// ---- POUs/XTS/Movers/VI_MoverVisu.TcVIS
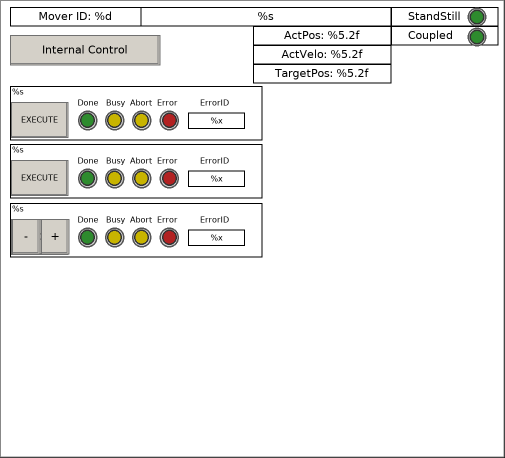
VISUALIZATION VI_MoverVisu  // 505x458
VAR_IN_OUT
	fbMover : FB_Mover;
END_VAR
    Rectangle (0,0 505x458)
    Rectangle (140,7 251x19), "%s", text variable: fbMover.ax.Status.MotionState, text list: 'AxisState_txt'
    Frame (10,86 252x54)
        shows VI_PLCOpenState(bExecute := fbMover.fbPower.Enable, sName := 'Power', bBusy := fbMover.fbPower.Busy, bDone := fbMover.fbPower.Status, bError := fbMover.fbPower.Error, bCommandAborted := fbMover.bTmp, ErrorID := fbMover.fbPower.ErrorID)
    Frame (10,144 252x54)
        shows VI_PLCOpenState(bExecute := fbMover.fbReset.Execute, sName := 'Reset', bBusy := fbMover.fbReset.Busy, bDone := fbMover.fbReset.Done, bError := fbMover.fbReset.Error, bCommandAborted := fbMover.bTmp, ErrorID := fbMover.fbReset.ErrorId)
    Button (10,35 150x30), "Internal Control", tooltip "Enable Visu Control, all methods will be locked"
        toggle fbMover.bInternalControl
    Rectangle (391,7 107x19), "StandStill"
    Lamp1 (466,6 22x22), variable: fbMover.ax.Status.StandStill, style: Lamp-Lamp1-Green
    Rectangle (10,7 131x19), "Mover ID: %d", text variable: fbMover.udiID
    Rectangle (253,26 138x19), "ActPos: %5.2f", text variable: fbMover.ax.NcToPlc.ModuloActPos, text list: 'AxisState_txt'
    Rectangle (253,45 138x19), "ActVelo: %5.2f", text variable: fbMover.ax.NcToPlc.ActVelo, text list: 'AxisState_txt'
    Rectangle (391,26 107x19), "Coupled"
    Lamp1 (466,26 22x22), variable: fbMover.ax.Status.Coupled, style: Lamp-Lamp1-Green
    Frame (10,203 252x54)
        shows VI_PLCOpenState(bExecute := fbMover.bTmp, sName := 'JogCA', bBusy := fbMover.fbJogCA.Busy, bDone := fbMover.fbJogCA.Done, bError := fbMover.fbJogCA.Error, bCommandAborted := fbMover.fbJogCA.CommandAborted, ErrorID := fbMover.fbJogCA.ErrorID)
    Button (12,219 28x35), "-"
        toggle fbMover.fbJogCA.JogBackwards
    Button (41,219 28x35), "+"
        toggle fbMover.fbJogCA.JogForward
    Rectangle (253,64 138x19), "TargetPos: %5.2f", text variable: fbMover.lrTargetPos, text list: 'AxisState_txt'
END_VISUALIZATION

// ---- POUs/XTS/Movers/VI_MoversVisu.TcVIS
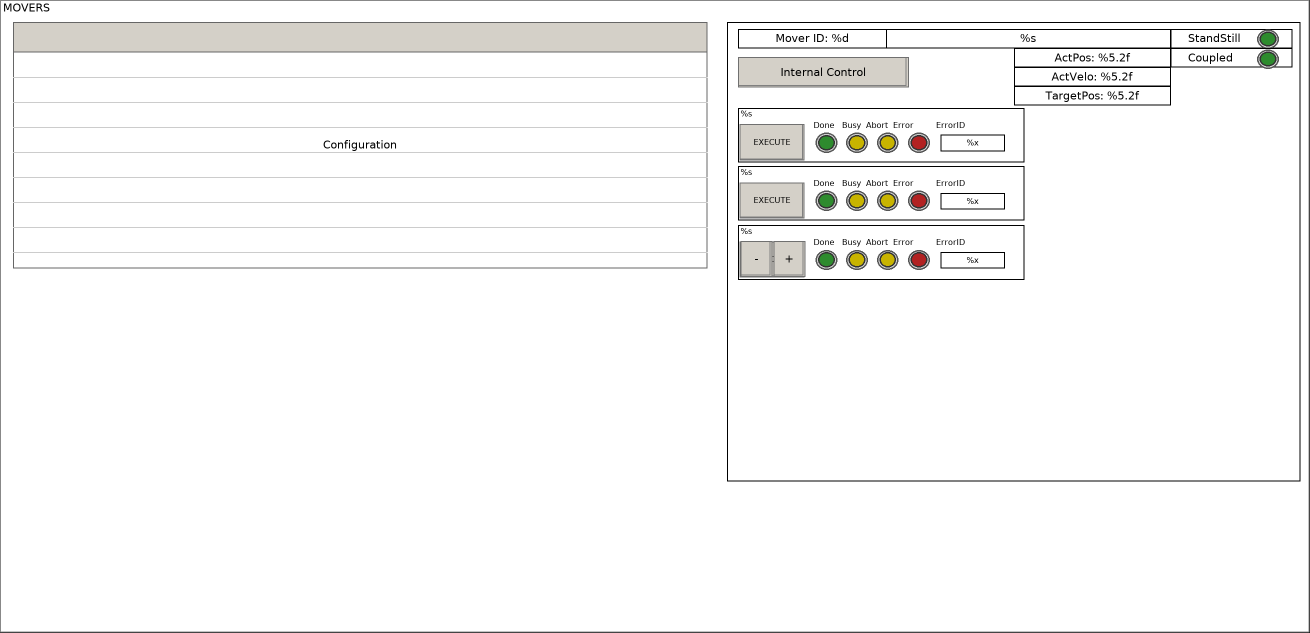
VISUALIZATION VI_MoversVisu  // 1310x633
VAR_IN_OUT
	ax		: ARRAY [1..Tc3_XTS_Utility.TcIoXtsEnvironmentParameterList.MaxXtsMoversPerXpu] OF FB_Mover;
END_VAR
VAR
	stTableStruct : ARRAY [1..25] OF stTableStructx10;
	iSelectedMover : INT;
END_VAR
    Rectangle (0,0 1310x633), "MOVERS"
    Frame (727,22 573x459), frame switch variable: iSelectedMover-1
        shows VI_MoverVisu(fbMover := ax[1])
        shows VI_MoverVisu(fbMover := ax[2])
        shows VI_MoverVisu(fbMover := ax[3])
        shows VI_MoverVisu(fbMover := ax[4])
        shows VI_MoverVisu(fbMover := ax[5])
        shows VI_MoverVisu(fbMover := ax[6])
        shows VI_MoverVisu(fbMover := ax[7])
        shows VI_MoverVisu(fbMover := ax[8])
        shows VI_MoverVisu(fbMover := ax[9])
        shows VI_MoverVisu(fbMover := ax[10])
        shows VI_MoverVisu(fbMover := ax[11])
        shows VI_MoverVisu(fbMover := ax[12])
        shows VI_MoverVisu(fbMover := ax[13])
        shows VI_MoverVisu(fbMover := ax[14])
        shows VI_MoverVisu(fbMover := ax[15])
        shows VI_MoverVisu(fbMover := ax[16])
        shows VI_MoverVisu(fbMover := ax[17])
        shows VI_MoverVisu(fbMover := ax[18])
        shows VI_MoverVisu(fbMover := ax[19])
        shows VI_MoverVisu(fbMover := ax[20])
        shows VI_MoverVisu(fbMover := ax[21])
        shows VI_MoverVisu(fbMover := ax[22])
        shows VI_MoverVisu(fbMover := ax[23])
        shows VI_MoverVisu(fbMover := ax[24])
        shows VI_MoverVisu(fbMover := ax[25])
    Table (13,22 694x246), "Configuration", data array: stTableStruct
        p1137915858: iSelectedMover
        p3854506369: ax[INDEX].ax.NcToPlc.AxisId
        p1892666644: ax[INDEX].ax.NcToPlc.ModuloSetPos
        p338671338: ax[INDEX].ax.NcToPlc.SetVelo
        p2170511999: ax[INDEX].ax.Status.MotionState
        p3723444502: ax[INDEX].ax.NcToPlc.ErrorCode
        p511219082: Position
        p1755163831: Velocity
        p2237128397: Error ID
        p505689113: Process Time
        p1757482276: Stop Positions
        p4088588272: Ack Mode
        p2243050616: Disable
        p516019884: Travel Time
        p2685023577: stTableStruct.b1
        p3312258591: stTableStruct.b2
        p1791247317: stTableStruct.b3
        p262371475: stTableStruct.b4
        p4008173056: stTableStruct.b5
        p2340480326: stTableStruct.b6
        p606709900: stTableStruct.b7
        p1095668682: stTableStruct.b8
        p1037165547: stTableStruct.b9
        p1488378029: stTableStruct.b10
        Columns.Column.[8].Template: xts.aStations[INDEX].stCfg.bDisable=true; toggle xts.aStations[INDEX].stCfg.bDisable
        Columns.Column.[6].Template: OnMouseClick: write the text variable via Default, min 1, max 3
        Columns.Column.[4].Template: OnMouseClick: write the text variable via Default
        Columns.Column.[5].Template: OnMouseClick: write the text variable via Default
        Columns.Column.[7].Template: OnMouseClick: write the text variable via Default
        Columns.Column.[9].Template: OnMouseClick: write the text variable via Default
END_VISUALIZATION

// ---- POUs/XTS/Stations/VI_StationVISU.TcVIS
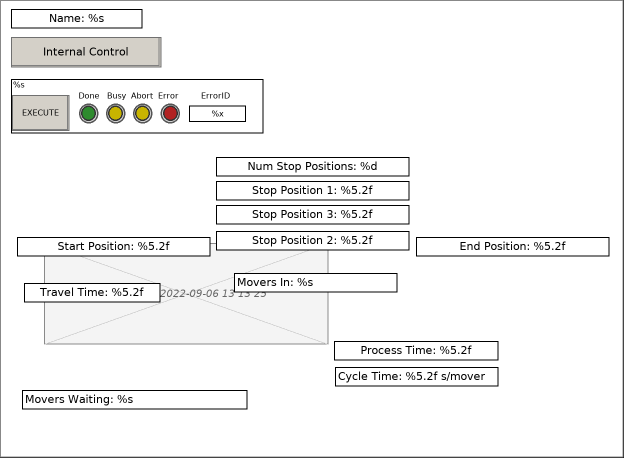
VISUALIZATION VI_StationVISU  // 624x458
VAR_IN_OUT
	fbStation : FB_Station;
END_VAR
    Rectangle (0,0 624x458)
    Frame (11,79 252x54)
        shows VI_PLCOpenState(bExecute := fbStation.bStart, sName := 'Secuence', bBusy := fbStation.stSecuenceStatus.bBusy, bDone := fbStation.stSecuenceStatus.bDone, bError := fbStation.stSecuenceStatus.bError, ErrorID := fbStation.stSecuenceStatus.udiErrorID)
    Button (11,37 150x30), "Internal Control", tooltip "Enable Visu Control, all methods will be locked"
        toggle fbStation.bInternalControl
    Rectangle (11,9 131x19), "Name: %s", text variable: fbStation.stCfg.sName
        OnMouseClick: write the text variable via Default
    Image (44,243 284x101), image: ImagePool.2022-09-06 13 13 25
    Rectangle (17,237 193x19), "Start Position: %5.2f", text variable: fbStation.stCfg.lrStartPosition
        OnMouseClick: write the text variable via Default
    Rectangle (416,237 193x19), "End Position: %5.2f", text variable: fbStation.stCfg.lrEndPosition
        OnMouseClick: write the text variable via Default
    Rectangle (234,273 163x19), "Movers In: %s", text variable: fbStation.sMoversIn
        OnMouseClick: write the text variable via Default
    Rectangle (22,390 225x19), "Movers Waiting: %s", text variable: fbStation.sMoversWaiting
        OnMouseClick: write the text variable via Default
    Rectangle (216,157 193x19), "Num Stop Positions: %d", text variable: fbStation.stCfg.uiNumStopPositions
        OnMouseClick: write the text variable via Default
    Rectangle (216,181 193x19), "Stop Position 1: %5.2f", text variable: fbStation.stCfg.lrStopPosition[1]
        OnMouseClick: write the text variable via Default
    Rectangle (216,231 193x19), "Stop Position 2: %5.2f", text variable: fbStation.stCfg.lrStopPosition[2], invisible if: fbStation.stCfg.uiNumStopPositions < 2
        OnMouseClick: write the text variable via Default
    Rectangle (216,205 193x19), "Stop Position 3: %5.2f", text variable: fbStation.stCfg.lrStopPosition[3], invisible if: fbStation.stCfg.uiNumStopPositions < 3
        OnMouseClick: write the text variable via Default
    Rectangle (335,367 163x19), "Cycle Time: %5.2f s/mover", text variable: (fbStation.lrActualProcessTime+fbStation.lrActualWaitingTime)/udint_to_lreal(fbStation.stCfg.uiNumStopPositions)
    Rectangle (24,283 136x19), "Travel Time: %5.2f", text variable: fbStation.stCfg.lrTravelTime
        OnMouseClick: write the text variable via Default
    Rectangle (334,341 164x19), "Process Time: %5.2f", text variable: fbStation.stCfg.lrProcessingTime
        OnMouseClick: write the text variable via Default
END_VISUALIZATION

// ---- POUs/XTS/Stations/VI_StationsVISU.TcVIS
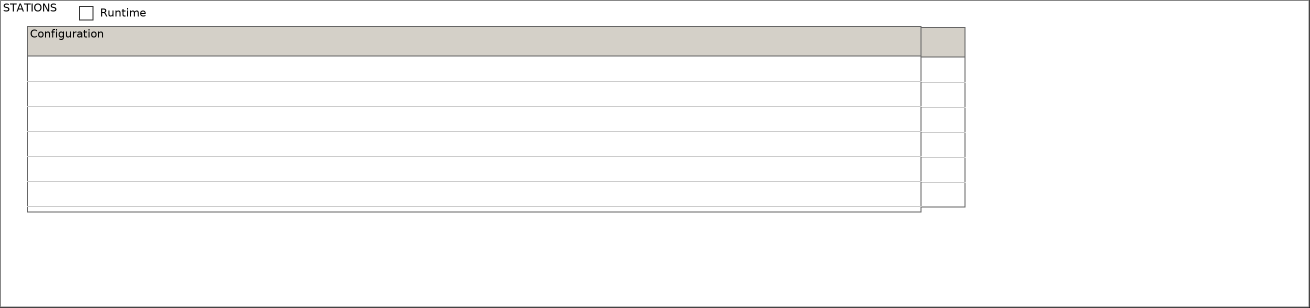
VISUALIZATION VI_StationsVISU  // 1310x308
VAR_IN_OUT
	aStations		: ARRAY [1..Tc3_XTS_Utility.TcIoXtsEnvironmentParameterList.MaxXtsInfoStation] OF FB_Station; //Stations
END_VAR
VAR
	stTableStruct : ARRAY [1..25] OF stTableStructx10;
	iSelectedStation : INT;
	bRunTime		: BOOL;
END_VAR
    Rectangle (0,0 1310x308), "STATIONS"
    Table (27,27 938x180), "Configuration", invisible if: bRunTime=true, data array: stTableStruct
        p1137915858: iSelectedStation
        p3854506369: aStations[INDEX].stCfg.sName
        p1892666644: aStations[INDEX].stCfg.lrStartPosition
        p338671338: aStations[INDEX].stCfg.lrStopPosition[1]
        p2170511999: aStations[INDEX].stCfg.lrStopPosition[2]
        p3723444502: aStations[INDEX].stCfg.lrStopPosition[3]
        p1218418051: aStations[INDEX].stCfg.lrProcessingTime
        p746581629: aStations[INDEX].stCfg.uiNumStopPositions
        p3104783080: aStations[INDEX].stCfg.lrTravelTime
        p7306298: aStations[INDEX].stCfg.lrEndPosition
        p511219082: Start Position
        p1755163831: Stop Position 1
        p4092479075: Stop Position 2
        p2237128397: Stop Position 3
        p505689113: Process Time
        p1757482276: Stop Positions
        p4088588272: Travel Time
        p2243050616: Extra Cfg.
        p516019884: End Position
        p2685023577: stTableStruct.b1
        p3312258591: stTableStruct.b2
        p1791247317: stTableStruct.b3
        p262371475: stTableStruct.b4
        p4008173056: stTableStruct.b5
        p2340480326: stTableStruct.b6
        p606709900: stTableStruct.b7
        p1095668682: stTableStruct.b8
        p1037165547: stTableStruct.b9
        p1488378029: stTableStruct.b10
        Columns.Column.[3].Template: OnMouseClick: write the text variable via Default
        Columns.Column.[6].Template: OnMouseClick: write the text variable via Default, min 1, max 3
        Columns.Column.[4].Template: OnMouseClick: write the text variable via Default
        Columns.Column.[5].Template: OnMouseClick: write the text variable via Default
        Columns.Column.[2].Template: OnMouseClick: write the text variable via Default
        Columns.Column.[7].Template: OnMouseClick: write the text variable via Default
        Columns.Column.[9].Template: OnMouseClick: write the text variable via Default
        Columns.Column.[1].Template: OnMouseClick: write the text variable via Default
    Checkbox (77,2 150x22), "Runtime", variable: bRunTime
    Table (27,26 894x186), "Configuration", invisible if: bRunTime=false, data array: stTableStruct
        p225073791: %5.2f s/m
        p3854506369: aStations[INDEX].stCfg.sName
        p1892666644: aStations[INDEX].stCfg.bEnableManualAck
        p338671338: aStations[INDEX].stCfg.bManualAck
        p2170511999: aStations[INDEX].fbMoversFIFO.nMovers
        p3723444502: aStations[INDEX].stCfg.udiSequenceState
        p1218418051: aStations[INDEX].udiErrorID
        p746581629: aStations[INDEX].sMoversWaiting
        p3104783080: aStations[INDEX].sMoversIn
        p2501879983: (aStations[INDEX].lrActualProcessTime+aStations[INDEX].lrActualWaitingTime)/udint_to_lreal(aStations[INDEX].stCfg.uiNumStopPositions)
        p7306298: xts.aStations[INDEX].lrActualWaitingTime
        p511219082: M. Ack
        p4092479075: Movers Waiting
        p505689113: Error ID
        p4088588272: Movers In
        p2243050616: Cycle Time
        p516019884: Waiting Time
        p2685023577: stTableStruct.b1
        p3312258591: stTableStruct.b2
        p1791247317: stTableStruct.b3
        p262371475: stTableStruct.b4
        p4008173056: stTableStruct.b5
        p2340480326: stTableStruct.b6
        p606709900: stTableStruct.b7
        p1095668682: stTableStruct.b8
        p1037165547: stTableStruct.b9
        p1488378029: stTableStruct.b10
        Columns.Column.[6].Template: OnMouseClick: write the text variable via Default, min 1, max 3
        Columns.Column.[4].Template: OnMouseClick: write the text variable via Default
        Columns.Column.[5].Template: OnMouseClick: write the text variable via Default
        Columns.Column.[2].Template: tap aStations[INDEX].stCfg.bManualAck
        Columns.Column.[0].Template: OnMouseClick: write the text variable via Default
        Columns.Column.[7].Template: OnMouseClick: write the text variable via Default
        Columns.Column.[9].Template: OnMouseClick: write the text variable via Default
        Columns.Column.[1].Template: toggle aStations[INDEX].stCfg.bEnableManualAck
END_VISUALIZATION

// ---- POUs/XTS/VISUs/TextList/AxisState_txt.TcTLO
TEXTLIST AxisState_txt
  0 = 'INVALID'
  1 = 'DISABLED'
  2 = 'STANDSTILL'
  3 = 'ERROR STOP'
  4 = 'STOPPING'
  5 = 'HOMING'
  6 = 'DISCRETE MOTION'
  7 = 'CONTINIOUS MOTION'
  8 = 'SYNCHRONIZED MOTION'
   = ''
END_TEXTLIST

// ---- POUs/XTS/VISUs/TextList/GroupState_txt.TcTLO
TEXTLIST GroupState_txt
  0 = 'INVALID'
  1 = 'DISABLED'
  2 = 'STANDBY'
  3 = 'MOVING'
  4 = 'STOPPING'
  5 = 'ERROR STOP'
  6 = 'HOMING'
  7 = 'NOT READY'
  8 = 'SUSPENDED'
   = ''
END_TEXTLIST

// ---- POUs/XTS/VISUs/TextList/MoversMode_txt.TcTLO
TEXTLIST MoversMode_txt
  1 = 'Single'
  2 = 'Double'
  3 = 'Triple'
   = ''
END_TEXTLIST

// ---- POUs/XTS/VISUs/TextList/PML_Modes_txt.TcTLO
TEXTLIST PML_Modes_txt
  0 = 'Undefined'
  1 = 'Production'
  2 = 'Manual'
   = ''
END_TEXTLIST

// ---- POUs/XTS/VISUs/VI_PLCOpenState.TcVIS
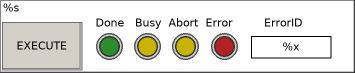
VISUALIZATION VI_PLCOpenState  // 355x73
VAR_IN_OUT
	bExecute : BOOL;	
END_VAR
VAR_INPUT
	sName	: STRING;
	bBusy : BOOL;
	bDone : BOOL;
	bError: BOOL;
	bCommandAborted : BOOL;
	ErrorID:UDINT;
END_VAR
    Rectangle (0,0 355x73), "%s", text variable: sName
    Lamp1 (94,31 31x31), variable: bDone, style: Lamp-Lamp1-Green
    Lamp1 (132,31 31x31), variable: bBusy, style: Lamp-Lamp1-Yellow
    Lamp1 (170,31 31x31), variable: bCommandAborted, style: Lamp-Lamp1-Yellow
    Lamp1 (209,31 31x31), variable: bError, style: Lamp-Lamp1-Red
    Rectangle (251,36 80x22), "%x", text variable: ErrorID
    Label (75,8 271x30), "Done Busy Abort Error ErrorID"
    Button (2,22 80x48), "EXECUTE"
        toggle bExecute
END_VISUALIZATION

// ---- POUs/XTS/VISUs/VI_XTSManualVisu.TcVIS
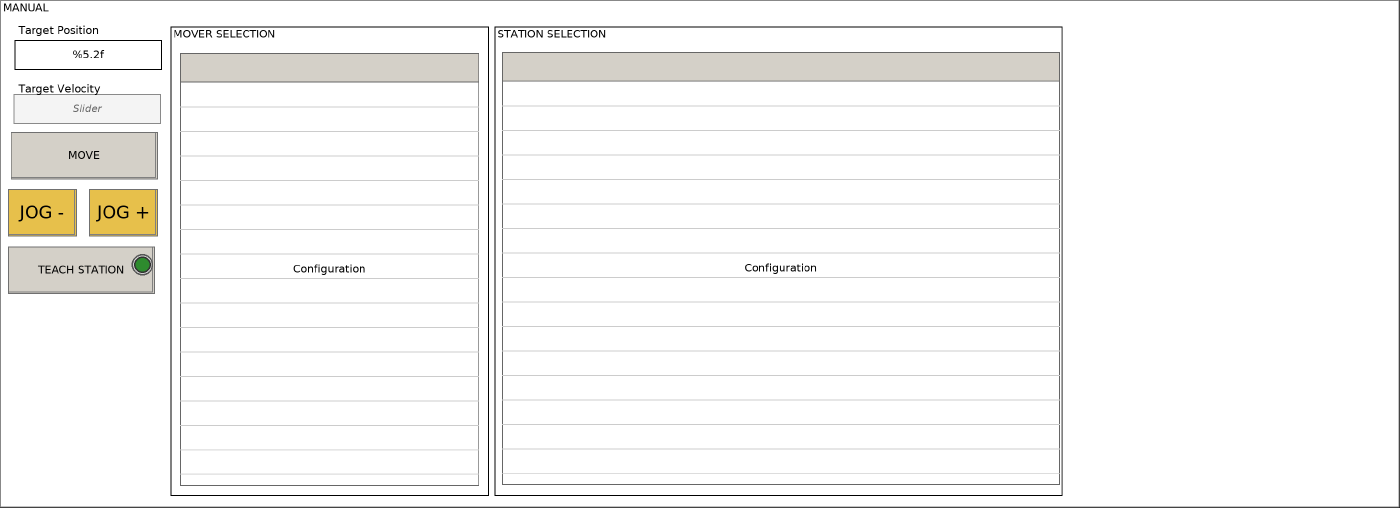
VISUALIZATION VI_XTSManualVisu  // 1430x519
VAR_IN_OUT
	xts : XTS_System;
END_VAR
VAR
	stTableStruct : ARRAY [1..20] OF stTableStructx10;
END_VAR
    Rectangle (0,0 1430x519), "MANUAL"
    Button (11,135 150x48), "MOVE"
        tap xts.bManualMove
    Slider (14,96 150x30), variable: xts.lrTargetVelocity, scale 1..4000
    Label (16,76 150x30), "Target Velocity"
    Rectangle (15,41 150x30), "%5.2f", text variable: xts.lrTargetPosition, input disabled if: xts.udiStationSelection<>0
        OnMouseClick: write the text variable via Default
    Label (16,16 150x30), "Target Position"
    Button (8,252 150x48), "TEACH STATION", input disabled if: xts.iVisuMoverSelection<1
        tap xts.bTeachStation
    Lamp1 (133,256 25x29), variable: xts.bTeachDone, style: Lamp-Lamp1-Green
    Rectangle (174,27 325x479), "MOVER SELECTION"
    Table (184,54 305x442), "Configuration", data array: stTableStruct
        p1137915858: xts.iVisuMoverSelection
        p3854506369: xts.ax[INDEX].ax.NcToPlc.AxisId
        p1892666644: xts.ax[INDEX].ax.NcToPlc.ModuloSetPos
        p338671338: xts.ax[INDEX].ax.NcToPlc.SetVelo
        p2170511999: xts.ax[INDEX].ax.Status.MotionState
        p3723444502: xts.ax[INDEX].ax.NcToPlc.ErrorCode
        p2232123230: Name
        p2685023577: stTableStruct.b1
        p511219082: Position
        p3312258591: stTableStruct.b2
        p1755163831: Velocity
        p1791247317: stTableStruct.b3
        p262371475: stTableStruct.b4
        p2237128397: Error ID
        p4008173056: stTableStruct.b5
        p505689113: Process Time
        p2340480326: stTableStruct.b6
        p1757482276: Stop Positions
        p606709900: stTableStruct.b7
        p4088588272: Ack Mode
        p1095668682: stTableStruct.b8
        p2243050616: Disable
        p1037165547: stTableStruct.b9
        p516019884: Travel Time
        p1488378029: stTableStruct.b10
        Columns.Column.[3].Template: OnMouseClick: write the text variable via Default
        Columns.Column.[9].Template: OnMouseClick: write the text variable via Default
        Columns.Column.[6].Template: OnMouseClick: write the text variable via Default, min 1, max 3
        Columns.Column.[5].Template: OnMouseClick: write the text variable via Default
        Columns.Column.[0].Template: OnMouseClick: OpenDialog Dialog=Mover_VISU, Parameters={fbMover: xts.aMovers[INDEX]}, OpenModal=True, OpenCentered=True
        Columns.Column.[8].Template: xts.aStations[INDEX].stCfg.bDisable=true; toggle xts.aStations[INDEX].stCfg.bDisable
        Columns.Column.[7].Template: OnMouseClick: write the text variable via Default
        Columns.Column.[4].Template: OnMouseClick: write the text variable via Default
    Rectangle (505,27 580x479), "STATION SELECTION"
    Table (513,53 569x442), "Configuration", data array: stTableStruct
        p1137915858: xts.iVisuStationSelection
        p1420305297: xts.iVisuStopPositionSelection
        p3854506369: xts.stCfg.stStationsCfg[INDEX].sName
        p1892666644: xts.stCfg.stStationsCfg[INDEX].lrStartPosition
        p338671338: xts.stCfg.stStationsCfg[INDEX].lrStopPosition[1]
        p2170511999: xts.stCfg.stStationsCfg[INDEX].lrStopPosition[2]
        p3723444502: xts.stCfg.stStationsCfg[INDEX].lrStopPosition[3]
        p1218418051: xts.stCfg.stStationsCfg[INDEX].lrProcessingTime
        p746581629: xts.stCfg.stStationsCfg[INDEX].uiNumStopPositions
        p3104783080: xts.stCfg.stStationsCfg[INDEX].lrTravelTime
        p7306298: xts.stCfg.stStationsCfg[INDEX].lrEndPosition
        p2685023577: stTableStruct.b1
        p511219082: Start Position
        p3312258591: stTableStruct.b2
        p1755163831: Stop Position 1
        p1791247317: stTableStruct.b3
        p4092479075: Stop Position 2
        p262371475: stTableStruct.b4
        p2237128397: Stop Position 3
        p4008173056: stTableStruct.b5
        p505689113: Process Time
        p2340480326: stTableStruct.b6
        p1757482276: Stop Positions
        p606709900: stTableStruct.b7
        p4088588272: Travel Time
        p1095668682: stTableStruct.b8
        p2243050616: Extra Cfg.
        p1037165547: stTableStruct.b9
        p516019884: End Position
        p1488378029: stTableStruct.b10
        Columns.Column.[6].Template: OnMouseClick: write the text variable via Default, min 1, max 3
        Columns.Column.[5].Template: OnMouseClick: write the text variable via Default
        Columns.Column.[7].Template: OnMouseClick: write the text variable via Default
    Button (8,193 70x48), "JOG -"
        tap xts.bJogBackwards
    Button (91,193 70x48), "JOG +"
        tap xts.bJogForward
END_VISUALIZATION

// ---- POUs/XTS/VISUs/VI_XTSMainVisu.TcVIS
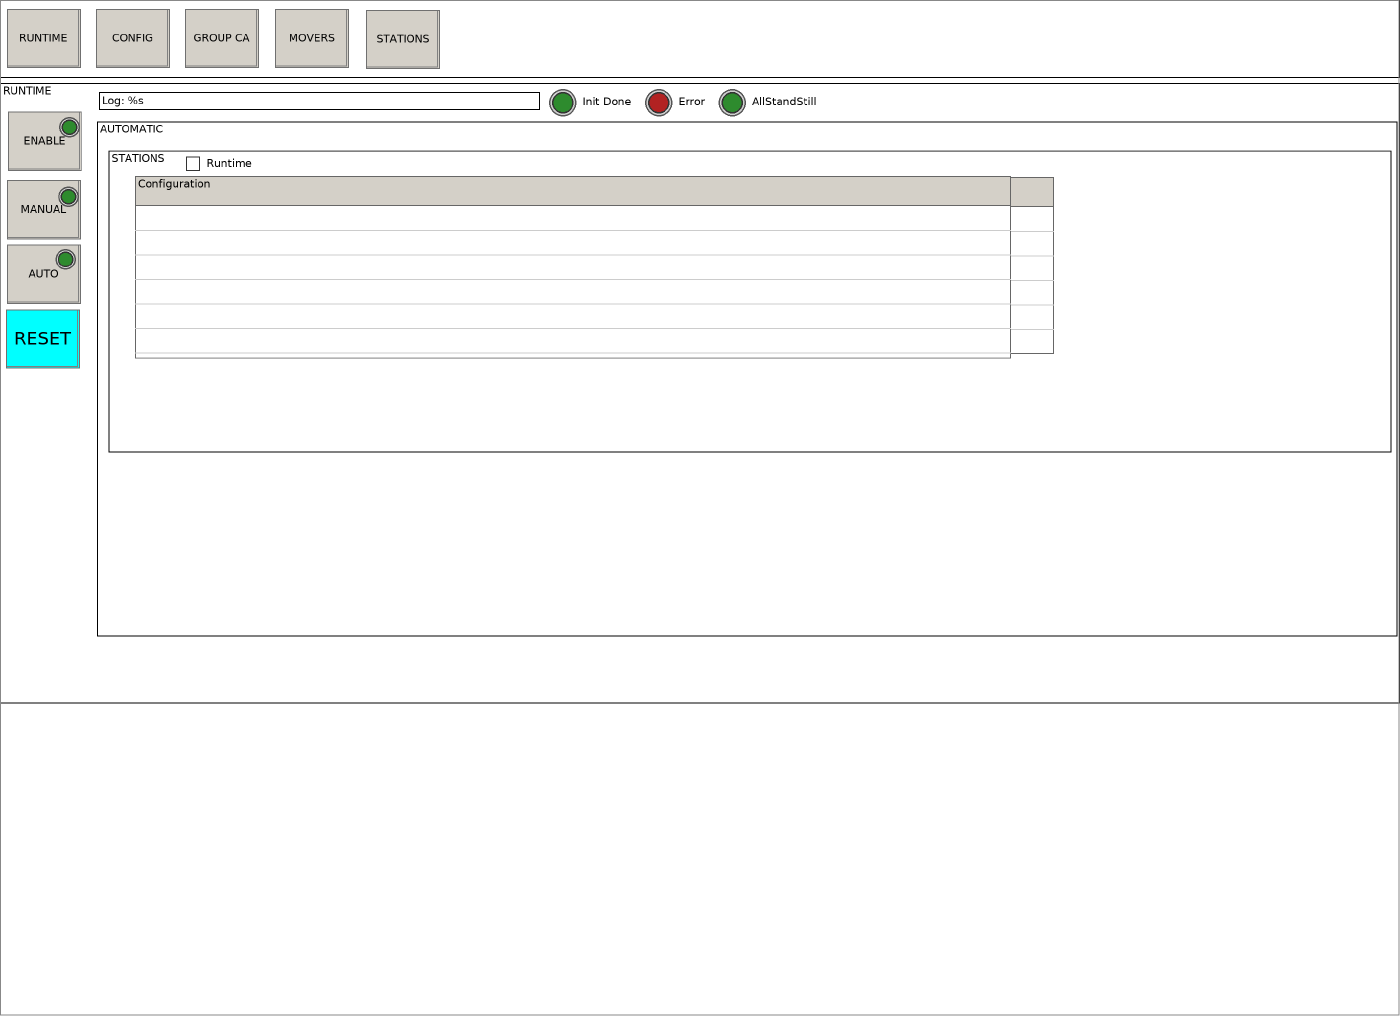
VISUALIZATION VI_XTSMainVisu  // 1430x1038
VAR_IN_OUT
	xts : XTS_System;
END_VAR
    Rectangle (0,0 1430x79)
    Button (7,9 75x60), "RUNTIME", colour toggle: xts.iFrameSelection=0
        OnMouseClick: execute { xts.iFrameSelection := 0; }
    Frame (0,85 1008x953), frame switch variable: xts.iFrameSelection
        shows VI_XTSRunTimeVisu(xts := xts)
        shows VI_XTSConfigurationVisu(xts := xts)
        shows VI_GroupCAVisu(gca := xts.gp)
        shows VI_MoversVisu(ax := xts.ax)
        shows VI_StationsVISU(aStations := xts.aStations)
    Button (98,9 75x60), "CONFIG", colour toggle: xts.iFrameSelection=1
        OnMouseClick: execute { xts.iFrameSelection := 1; }
    Button (189,9 75x60), "GROUP CA", colour toggle: xts.iFrameSelection=2
        OnMouseClick: execute { xts.iFrameSelection := 2; }
    Button (281,9 75x60), "MOVERS", colour toggle: xts.iFrameSelection=3
        OnMouseClick: execute { xts.iFrameSelection := 3; }
    Button (374,10 75x60), "STATIONS", colour toggle: xts.iFrameSelection=4
        OnMouseClick: execute { xts.iFrameSelection := 4; }
END_VISUALIZATION

// ---- POUs/XTS/VISUs/VI_XTSRunTimeVisu.TcVIS
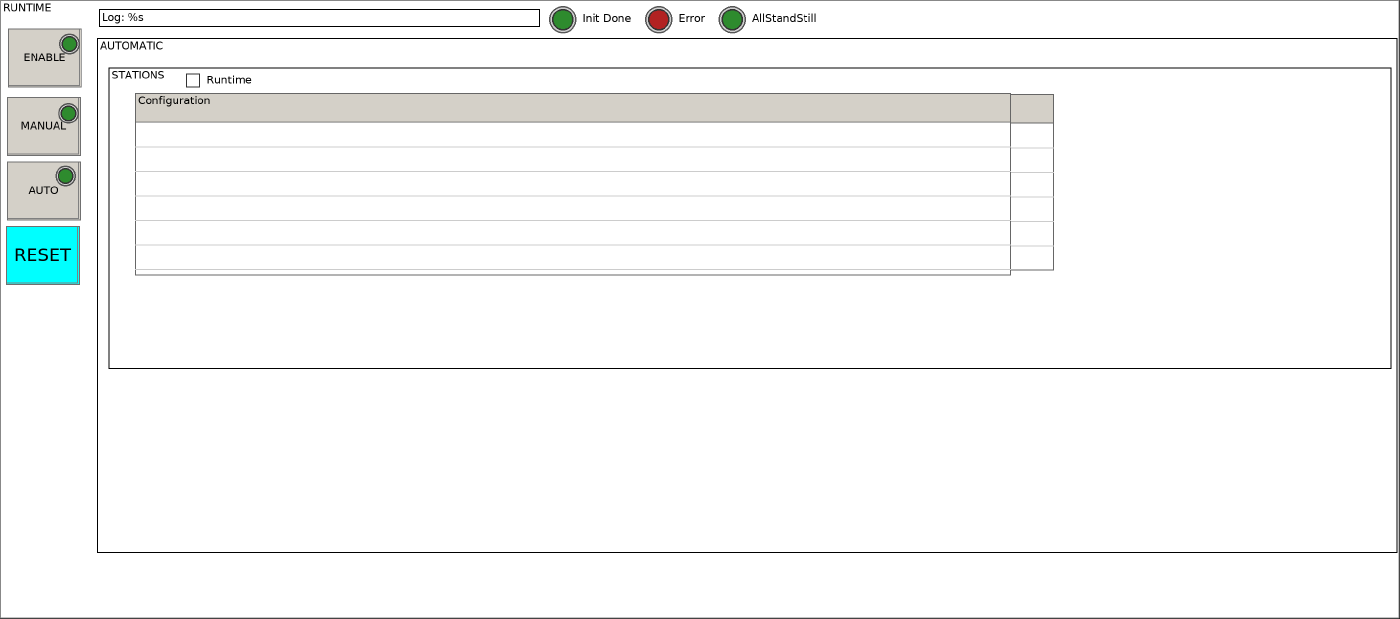
VISUALIZATION VI_XTSRunTimeVisu  // 1430x633
VAR_IN_OUT
	xts : XTS_System;
END_VAR
    Rectangle (0,0 1430x633), "RUNTIME"
    Button (8,29 75x60), "ENABLE"
        toggle xts.bEnable
    Button (7,99 75x60), "MANUAL", input disabled if: xts.bInAutomatic = TRUE
        toggle xts.bManual
        OnMouseClick: FrameSelectionChange Selection=SelectedFrame=a18850ea-e303-4efa-b84e-5057b211b999, Selection=1, GlobSel=AssignType=Directly, SelType=Locally
    Button (7,165 75x60), "AUTO", input disabled if: xts.bInManual = TRUE
        toggle xts.bAutomatic
        OnMouseClick: FrameSelectionChange Selection=SelectedFrame=a18850ea-e303-4efa-b84e-5057b211b999, GlobSel=AssignType=Directly, SelType=Locally
    Lamp1 (559,4 32x32), variable: xts.bInitDone, style: Lamp-Lamp1-Green
    Label (592,4 110x30), "Init Done"
    Lamp1 (657,4 32x32), variable: xts.bError, style: Lamp-Lamp1-Red
    Label (690,4 110x30), "Error"
    Lamp1 (732,4 32x32), variable: xts.bAllMoversStandStill, style: Lamp-Lamp1-Green
    Label (765,4 110x30), "AllStandStill"
    Lamp1 (59,32 24x26), variable: xts.bEnabled, style: Lamp-Lamp1-Green
    Rectangle (101,9 450x18), "Log: %s", text variable: xts.sLog
        OnMouseClick: write the text variable via Default
    Frame (99,39 1317x468)
        shows VI_XTSAutoVisu(xts := xts)
        shows VI_XTSManualVisu(xts := xts)
    Lamp1 (55,167 24x26), variable: xts.bInAutomatic=true, style: Lamp-Lamp1-Green
    Lamp1 (58,103 24x26), variable: xts.bInManual=true, style: Lamp-Lamp1-Green
    Button (6,231 75x60), "RESET"
        tap xts.bReset
END_VISUALIZATION

// ---- POUs/XTS/VISUs/VI_XTSConfigurationVisu.TcVIS
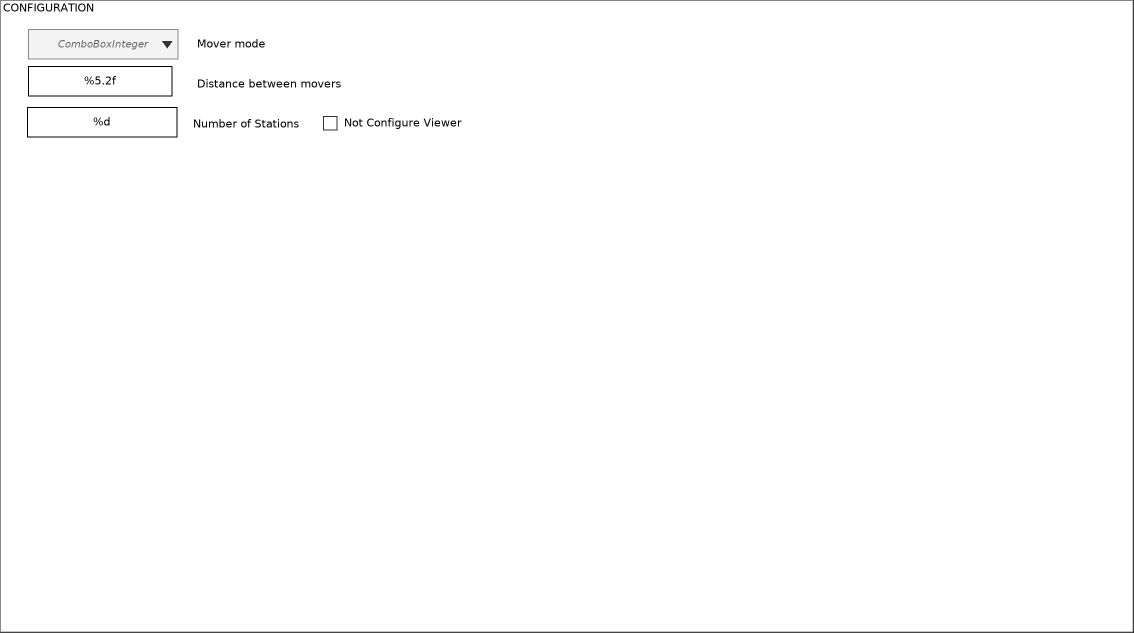
VISUALIZATION VI_XTSConfigurationVisu  // 1134x633
VAR_IN_OUT
	xts : XTS_System;
END_VAR
VAR
	stTableStruct : ARRAY [1..25] OF stTableStructx10;
END_VAR
    Rectangle (0,0 1134x633), "CONFIGURATION"
    Rectangle (27,107 150x30), "%d", text variable: xts.stCfg.udiNumStations
        OnMouseClick: write the text variable via Default
    Label (190,109 150x30), "Number of Stations"
    Checkbox (321,108 165x30), "Not Configure Viewer", variable: xts.stCfg.bNotCfgStationsViewer
    Label (194,29 150x30), "Mover mode"
    ComboBoxInteger (28,29 150x30), variable: xts.stCfg.udiMoverMode, text list: 'MoverMode_TXT'
    Label (194,69 150x30), "Distance between movers"
    Rectangle (28,66 144x30), "%5.2f", text variable: xts.stCfg.lrMoverDistance
        OnMouseClick: write the text variable via Default
END_VISUALIZATION

// ---- POUs/XTS/VISUs/VI_XTSAutoVisu.TcVIS
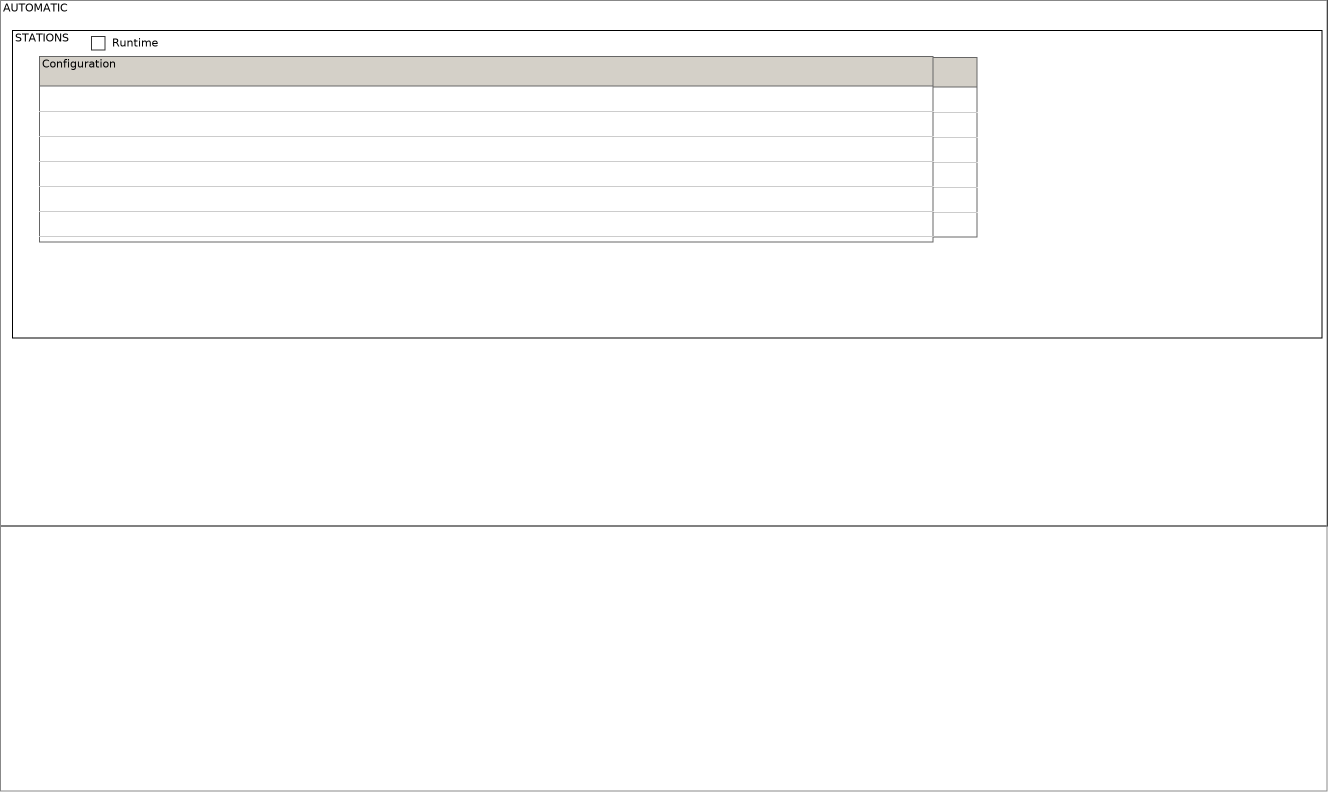
VISUALIZATION VI_XTSAutoVisu  // 1328x792
VAR_IN_OUT
	xts : XTS_System;
END_VAR
VAR
	stTableStruct : ARRAY [1..25] OF stTableStructx10;
END_VAR
    Rectangle (0,0 1328x526), "AUTOMATIC"
    Frame (12,30 1311x762)
        shows VI_StationsVISU(aStations := xts.aStations)
END_VISUALIZATION

// ---- VISUs/MAIN_VISU.TcVIS
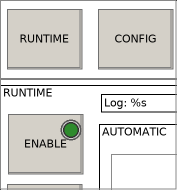
VISUALIZATION MAIN_VISU  // 177x190
    Frame (0,0 177x190)
        shows VI_XTSMainVisu(xts := XTS_PRG.fbXTSSystem)
END_VISUALIZATION
